(* PLC project marvel_vessel, Institute of Astronomy Onto 0.0.1 *)
(* stored: creationDateTime 2025-01-01T00:00:00.0, modificationDateTime 2025-01-01T00:00:00.0 *)

TYPE heaterControlProcesses : STRUCT
  {attribute 'TcHmiSymbol.Show'}
  start : Process;  (* Start warming up *)
  {attribute 'TcHmiSymbol.Show'}
  stop : Process;  (* Stop heating *)
  {attribute 'TcHmiSymbol.Show'}
  reset : Process;  (* Reset any errors *)
END_STRUCT;
END_TYPE

TYPE vesselProcesses : STRUCT
  {attribute 'TcHmiSymbol.Show'}
  initialize : Process;  (* Start initializing *)
  {attribute 'TcHmiSymbol.Show'}
  start : Process;  (* Start warming up *)
  {attribute 'TcHmiSymbol.Show'}
  stop : Process;  (* Stop all temperature control and heating *)
  {attribute 'TcHmiSymbol.Show'}
  reset : Process;  (* Reset any errors *)
END_STRUCT;
END_TYPE

TYPE temperatureMeasurementStatuses : STRUCT
  {attribute 'OPC.UA.DA' := '1'}
  {attribute 'OPC.UA.DA.Access' := '1'}
  {attribute 'TcHmiSymbol.Show'}
  enabled : EnabledStatus;  (* Is the temperature being measured? *)
  {attribute 'OPC.UA.DA' := '1'}
  {attribute 'OPC.UA.DA.Access' := '1'}
  {attribute 'TcHmiSymbol.Show'}
  health : HealthStatus;  (* Is the measurement OK? *)
  {attribute 'OPC.UA.DA' := '1'}
  {attribute 'OPC.UA.DA.Access' := '1'}
  {attribute 'TcHmiSymbol.Show'}
  alarm : HiHiLoLoAlarmStatus;  (* Alarm status *)
END_STRUCT;
END_TYPE

TYPE heaterControlStatuses : STRUCT
  {attribute 'OPC.UA.DA' := '1'}
  {attribute 'OPC.UA.DA.Access' := '1'}
  {attribute 'TcHmiSymbol.Show'}
  enabled : EnabledStatus;  (* Is the heater enabled? *)
  {attribute 'OPC.UA.DA' := '1'}
  {attribute 'OPC.UA.DA.Access' := '1'}
  {attribute 'TcHmiSymbol.Show'}
  health : HealthStatus;  (* Is the heater healthy? *)
  {attribute 'OPC.UA.DA' := '1'}
  {attribute 'OPC.UA.DA.Access' := '1'}
  {attribute 'TcHmiSymbol.Show'}
  busy : BusyStatus;  (* Is the heater busy (e.g. ramping)? *)
END_STRUCT;
END_TYPE

TYPE vesselStatuses : STRUCT
  {attribute 'OPC.UA.DA' := '1'}
  {attribute 'OPC.UA.DA.Access' := '1'}
  {attribute 'TcHmiSymbol.Show'}
  init : InitializationStatus;
  {attribute 'OPC.UA.DA' := '1'}
  {attribute 'OPC.UA.DA.Access' := '1'}
  {attribute 'TcHmiSymbol.Show'}
  health : HealthStatus;
  {attribute 'OPC.UA.DA' := '1'}
  {attribute 'OPC.UA.DA.Access' := '1'}
  {attribute 'TcHmiSymbol.Show'}
  busy : BusyStatus;
END_STRUCT;
END_TYPE

TYPE vesselHeaterConfig : STRUCT
  {attribute 'TcHmiSymbol.Show'}
  name : STRING;  (* Name of the heater *)
  {attribute 'TcHmiSymbol.Show'}
  enabled : BOOL;  (* True if the heater is enabled *)
  {attribute 'TcHmiSymbol.Show'}
  setPoint : REAL;  (* set point temperature in kelvin *)
  {attribute 'TcHmiSymbol.Show'}
  fastHeatingSetPoint : REAL;  (* set point temperature in kelvin used for fast heating (e.g. during ramping) *)
  {attribute 'TcHmiSymbol.Show'}
  maxPower : REAL;  (* Maximum power of the heater *)
  {attribute 'TcHmiSymbol.Show'}
  p : REAL;  (* proportional gain *)
  {attribute 'TcHmiSymbol.Show'}
  i : REAL;  (* integral gain *)
  {attribute 'TcHmiSymbol.Show'}
  d : REAL;  (* derivative gain *)
  {attribute 'TcHmiSymbol.Show'}
  weightTemperatureSensors : ARRAY[0..25] OF REAL;  (* value between 0-1 representing the weight of each temperature sensor (0 for sensors not effecting this heater) *)
END_STRUCT;
END_TYPE

TYPE vesselTemperatureSensorConfig : STRUCT
  {attribute 'TcHmiSymbol.Show'}
  name : STRING;  (* Name of the temperature sensor *)
  {attribute 'TcHmiSymbol.Show'}
  enabled : BOOL;  (* Is the quantity being measured? (Can be false e.g. if the sensor is deliberately not connected (yet).) *)
  {attribute 'TcHmiSymbol.Show'}
  gain : LREAL := 1.0;  (* Gain to be applied to the measured value (default: 1 = no gain) *)
  {attribute 'TcHmiSymbol.Show'}
  offset : LREAL;  (* Offset to be added to the measured value (default: 0 = no offset) *)
  {attribute 'TcHmiSymbol.Show'}
  alarms : HiHiLoLoAlarmConfig;  (* Config *)
END_STRUCT;
END_TYPE

TYPE vesselConfig : STRUCT
  {attribute 'TcHmiSymbol.Show'}
  setPointTarger : REAL;  (* set point temperature in kelvin *)
  {attribute 'TcHmiSymbol.Show'}
  rampVeloPos : REAL;  (* velocity of temperature change in K/s while ramping up *)
  {attribute 'TcHmiSymbol.Show'}
  rampVeloNeg : REAL;  (* velocity of temperature change in K/s while ramping down *)
END_STRUCT;
END_TYPE

TYPE M_SM_temperatureMeasurement : STRUCT
  {attribute 'OPC.UA.DA' := '1'}
  {attribute 'OPC.UA.DA.Access' := '1'}
  {attribute 'TcHmiSymbol.Show'}
  actualStatus : STRING;
  {attribute 'OPC.UA.DA' := '1'}
  {attribute 'OPC.UA.DA.Access' := '1'}
  {attribute 'TcHmiSymbol.Show'}
  actual : Temperature;
  {attribute 'OPC.UA.DA' := '1'}
  {attribute 'OPC.UA.DA.Access' := '1'}
  {attribute 'TcHmiSymbol.Show'}
  average : Temperature;
  {attribute 'OPC.UA.DA' := '1'}
  {attribute 'OPC.UA.DA.Access' := '1'}
  {attribute 'TcHmiSymbol.Show'}
  underrange : BOOL;
  {attribute 'OPC.UA.DA' := '1'}
  {attribute 'OPC.UA.DA.Access' := '1'}
  {attribute 'TcHmiSymbol.Show'}
  overrange : BOOL;
  {attribute 'OPC.UA.DA' := '1'}
  {attribute 'TcHmiSymbol.Show'}
  stat : temperatureMeasurementStatuses;
END_STRUCT;
END_TYPE

TYPE M_SM_heaterControl : STRUCT
  {attribute 'OPC.UA.DA' := '1'}
  {attribute 'OPC.UA.DA.Access' := '1'}
  {attribute 'TcHmiSymbol.Show'}
  actualStatus : STRING;
  {attribute 'OPC.UA.DA' := '1'}
  {attribute 'OPC.UA.DA.Access' := '1'}
  {attribute 'TcHmiSymbol.Show'}
  setPointRamped : REAL;
  {attribute 'OPC.UA.DA' := '1'}
  {attribute 'OPC.UA.DA.Access' := '1'}
  {attribute 'TcHmiSymbol.Show'}
  power : REAL;
  {attribute 'OPC.UA.DA' := '1'}
  {attribute 'OPC.UA.DA.Access' := '1'}
  {attribute 'TcHmiSymbol.Show'}
  associatedTemperature : REAL;
  {attribute 'OPC.UA.DA' := '1'}
  {attribute 'OPC.UA.DA.Access' := '1'}
  {attribute 'TcHmiSymbol.Show'}
  setPointDeviation : REAL;
  {attribute 'OPC.UA.DA' := '1'}
  {attribute 'OPC.UA.DA.Access' := '1'}
  {attribute 'TcHmiSymbol.Show'}
  isControlled : BOOL;
  {attribute 'OPC.UA.DA' := '1'}
  {attribute 'TcHmiSymbol.Show'}
  stat : heaterControlStatuses;
  {attribute 'OPC.UA.DA' := '1'}
  {attribute 'TcHmiSymbol.Show'}
  proc : M_SM_heaterControlProcesses;
END_STRUCT;
END_TYPE

TYPE M_SM_vessel : STRUCT
  {attribute 'OPC.UA.DA' := '1'}
  {attribute 'OPC.UA.DA.Access' := '1'}
  {attribute 'TcHmiSymbol.Show'}
  actualStatus : STRING;
  {attribute 'OPC.UA.DA' := '1'}
  {attribute 'OPC.UA.DA.Access' := '1'}
  {attribute 'TcHmiSymbol.Show'}
  config : vesselConfig;
  {attribute 'OPC.UA.DA' := '1'}
  {attribute 'OPC.UA.DA.Access' := '1'}
  {attribute 'TcHmiSymbol.Show'}
  isControlled : BOOL;
  {attribute 'OPC.UA.DA' := '1'}
  {attribute 'OPC.UA.DA.Access' := '1'}
  {attribute 'TcHmiSymbol.Show'}
  setPointRamped : REAL;
  {attribute 'OPC.UA.DA' := '1'}
  {attribute 'OPC.UA.DA.Access' := '1'}
  {attribute 'TcHmiSymbol.Show'}
  temperatureSensor : ARRAY[0..25] OF temperatureMeasurement;
  {attribute 'OPC.UA.DA' := '1'}
  {attribute 'OPC.UA.DA.Access' := '1'}
  {attribute 'TcHmiSymbol.Show'}
  vesselHeater : ARRAY[0..25] OF heaterControl;
  {attribute 'OPC.UA.DA' := '1'}
  {attribute 'TcHmiSymbol.Show'}
  stat : vesselStatuses;
  {attribute 'OPC.UA.DA' := '1'}
  {attribute 'TcHmiSymbol.Show'}
  proc : M_SM_vesselProcesses;
END_STRUCT;
END_TYPE

TYPE M_SM_heaterControlProcesses : STRUCT
  {attribute 'TcHmiSymbol.Show'}
  start : M_Process;
  {attribute 'TcHmiSymbol.Show'}
  stop : M_Process;
  {attribute 'TcHmiSymbol.Show'}
  reset : M_Process;
END_STRUCT;
END_TYPE

TYPE M_SM_vesselProcesses : STRUCT
  {attribute 'TcHmiSymbol.Show'}
  initialize : M_Process;
  {attribute 'TcHmiSymbol.Show'}
  start : M_Process;
  {attribute 'TcHmiSymbol.Show'}
  stop : M_Process;
  {attribute 'TcHmiSymbol.Show'}
  reset : M_Process;
END_STRUCT;
END_TYPE

FUNCTION_BLOCK SM_temperatureMeasurement
  VAR_INPUT
    {attribute 'OPC.UA.DA' := '0'}
    rawValue AT %I* : INT;  (* Measured raw value *)
    {attribute 'OPC.UA.DA' := '0'}
    error AT %I* : BOOL;  (* Error *)
    {attribute 'OPC.UA.DA' := '0'}
    conversionFactor : LREAL := 0.01;  (* rawValue * conversionFactor = temperature.degrees.value *)
  END_VAR
  VAR_OUTPUT
    {attribute 'OPC.UA.DA' := '1'}
    {attribute 'OPC.UA.DA.Access' := '1'}
    actualStatus : STRING(50);  (* Current status description *)
    {attribute 'OPC.UA.DA' := '1'}
    {attribute 'OPC.UA.DA.Access' := '1'}
    actual : Temperature;  (* Actual value *)
    {attribute 'OPC.UA.DA' := '1'}
    {attribute 'OPC.UA.DA.Access' := '1'}
    average : Temperature;  (* Moving average value *)
    {attribute 'OPC.UA.DA' := '1'}
    {attribute 'OPC.UA.DA.Access' := '1'}
    underrange AT %I* : BOOL;  (* Underrange *)
    {attribute 'OPC.UA.DA' := '1'}
    {attribute 'OPC.UA.DA.Access' := '1'}
    overrange AT %I* : BOOL;  (* Overrange *)
    {attribute 'OPC.UA.DA' := '1'}
    stat : temperatureMeasurementStatuses;  (* Statuses of the state machine *)
  END_VAR
  VAR_IN_OUT
    {attribute 'OPC.UA.DA' := '0'}
    config : vesselTemperatureSensorConfig;  (* Reference to the config (alarms in degrees celsius) *)
    {attribute 'OPC.UA.DA' := '0'}
    activity_ref : ActivityStatus;  (* Shared activity status *)
    {attribute 'OPC.UA.DA' := '0'}
    services_ref : Services;  (* Shared services *)
  END_VAR

            stat.enabled := F_EnabledStatus(
    superState := TRUE,
    isEnabled := config.enabled);
stat.health := F_HealthStatus(
    superState := stat.enabled = EnabledStatus.enabled,
    isGood := NOT(error OR (underrange OR (overrange OR ((stat.alarm = HiHiLoLoAlarmStatus.hiHi) OR (stat.alarm = HiHiLoLoAlarmStatus.loLo))))),
    hasWarning := (stat.alarm = HiHiLoLoAlarmStatus.hi) OR (stat.alarm = HiHiLoLoAlarmStatus.lo));
stat.alarm := F_HiHiLoLoAlarmStatus(
    superState := stat.enabled = EnabledStatus.enabled,
    config := config.alarms,
    value := average.celsius.value);

          

METHOD _copyFromModel_SM_temperatureMeasurement
  VAR_IN_OUT
    {attribute 'OPC.UA.DA' := '0'}
    model : M_SM_temperatureMeasurement;
  END_VAR
                  
                
END_METHOD

METHOD _copyToModel_SM_temperatureMeasurement
  VAR_IN_OUT
    {attribute 'OPC.UA.DA' := '0'}
    model : M_SM_temperatureMeasurement;
  END_VAR
                  model.actualStatus := THIS^.actualStatus;
model.actual := THIS^.actual;
model.average := THIS^.average;
model.underrange := THIS^.underrange;
model.overrange := THIS^.overrange;
model.stat := THIS^.stat;

                
END_METHOD
END_FUNCTION_BLOCK

FUNCTION_BLOCK SM_heaterControl
  VAR_OUTPUT
    {attribute 'OPC.UA.DA' := '1'}
    {attribute 'OPC.UA.DA.Access' := '1'}
    actualStatus : STRING(50);  (* Current status description *)
    {attribute 'OPC.UA.DA' := '1'}
    {attribute 'OPC.UA.DA.Access' := '1'}
    setPointRamped : REAL;  (* Set point temperature in kelvin *)
    {attribute 'OPC.UA.DA' := '1'}
    {attribute 'OPC.UA.DA.Access' := '1'}
    power : REAL;  (* Current power of the heater in percentage *)
    {attribute 'OPC.UA.DA' := '1'}
    {attribute 'OPC.UA.DA.Access' := '1'}
    associatedTemperature : REAL;  (* Temperature associated with the heater *)
    {attribute 'OPC.UA.DA' := '1'}
    {attribute 'OPC.UA.DA.Access' := '1'}
    setPointDeviation : REAL;  (* Current error between set point and associated temperature *)
    {attribute 'OPC.UA.DA' := '1'}
    {attribute 'OPC.UA.DA.Access' := '1'}
    isControlled : BOOL;  (* True if the heater is in controlled state *)
    {attribute 'OPC.UA.DA' := '1'}
    stat : heaterControlStatuses;  (* Statuses of the state machine *)
    {attribute 'OPC.UA.DA' := '1'}
    proc : heaterControlProcesses;  (* Processes of the state machine *)
  END_VAR
  VAR_IN_OUT
    {attribute 'OPC.UA.DA' := '0'}
    config : vesselHeaterConfig;  (* Reference to the heater config *)
    {attribute 'OPC.UA.DA' := '0'}
    activity_ref : ActivityStatus;  (* Shared activity status *)
    {attribute 'OPC.UA.DA' := '0'}
    services_ref : Services;  (* Shared services *)
  END_VAR

            stat.enabled := F_EnabledStatus(
    superState := TRUE,
    isEnabled := config.enabled);
stat.health := F_HealthStatus( superState := TRUE );
stat.busy := F_BusyStatus(
    superState := TRUE,
    isBusy := proc.start.stat.busy);
proc.start( isEnabled := config.enabled );
proc.stop();
proc.reset();

          

METHOD _copyFromModel_SM_heaterControl
  VAR_IN_OUT
    {attribute 'OPC.UA.DA' := '0'}
    model : M_SM_heaterControl;
  END_VAR
                  THIS^.proc.start._copyFromModel_Process( model := model.proc.start );
THIS^.proc.stop._copyFromModel_Process( model := model.proc.stop );
THIS^.proc.reset._copyFromModel_Process( model := model.proc.reset );

                
END_METHOD

METHOD _copyToModel_SM_heaterControl
  VAR_IN_OUT
    {attribute 'OPC.UA.DA' := '0'}
    model : M_SM_heaterControl;
  END_VAR
                  model.actualStatus := THIS^.actualStatus;
model.setPointRamped := THIS^.setPointRamped;
model.power := THIS^.power;
model.associatedTemperature := THIS^.associatedTemperature;
model.setPointDeviation := THIS^.setPointDeviation;
model.isControlled := THIS^.isControlled;
model.stat := THIS^.stat;
THIS^.proc.start._copyToModel_Process( model := model.proc.start );
THIS^.proc.stop._copyToModel_Process( model := model.proc.stop );
THIS^.proc.reset._copyToModel_Process( model := model.proc.reset );

                
END_METHOD
END_FUNCTION_BLOCK

FUNCTION_BLOCK SM_vessel
  VAR_OUTPUT
    {attribute 'OPC.UA.DA' := '1'}
    {attribute 'OPC.UA.DA.Access' := '1'}
    actualStatus : STRING(50);  (* Current status description *)
    {attribute 'OPC.UA.DA' := '1'}
    {attribute 'OPC.UA.DA.Access' := '1'}
    config : vesselConfig;  (* Active configuration of the vessel *)
    {attribute 'OPC.UA.DA' := '1'}
    {attribute 'OPC.UA.DA.Access' := '1'}
    isControlled : BOOL;  (* True if the vessel is in controlled state *)
    {attribute 'OPC.UA.DA' := '1'}
    {attribute 'OPC.UA.DA.Access' := '1'}
    setPointRamped : REAL;  (* Set point temperature in kelvin after ramping *)
    {attribute 'OPC.UA.DA' := '1'}
    {attribute 'OPC.UA.DA.Access' := '1'}
    temperatureSensor : ARRAY[0..25] OF temperatureMeasurement;  (* All vessel temperature sensors *)
    {attribute 'OPC.UA.DA' := '1'}
    {attribute 'OPC.UA.DA.Access' := '1'}
    vesselHeater : ARRAY[0..25] OF heaterControl;  (* All vessel heaters *)
    {attribute 'OPC.UA.DA' := '1'}
    stat : vesselStatuses;  (* Statuses of the state machine *)
    {attribute 'OPC.UA.DA' := '1'}
    proc : vesselProcesses;  (* Processes of the state machine *)
  END_VAR
  VAR_IN_OUT
    {attribute 'OPC.UA.DA' := '0'}
    activity_ref : ActivityStatus;  (* Shared activity status *)
    {attribute 'OPC.UA.DA' := '0'}
    services_ref : Services;  (* Shared services *)
    {attribute 'OPC.UA.DA' := '0'}
    config_ref : vesselConfig;  (* Active configuration of the vessel *)
  END_VAR

            stat.health := F_HealthStatus(
    superState := TRUE,
    isGood := ((stat.health = HealthStatus.good) OR (stat.health = HealthStatus.warning)) AND ((stat.health = HealthStatus.good) OR (stat.health = HealthStatus.warning)));
proc.initialize( isEnabled := (NOT(stat.init = InitializationStatus.locked)) AND ((stat.init = InitializationStatus.shutdown) OR ((stat.init = InitializationStatus.initializingFailed) OR (stat.init = InitializationStatus.initialized))) );
proc.start( isEnabled := (stat.init = InitializationStatus.initializingFailed) AND (stat.init = InitializationStatus.initialized) );
proc.stop( isEnabled := (stat.busy = BusyStatus.busy) OR isControlled );
proc.reset( isEnabled := (stat.busy = BusyStatus.idle) AND (stat.init = InitializationStatus.initialized) );

          

METHOD _copyFromModel_SM_vessel
  VAR_IN_OUT
    {attribute 'OPC.UA.DA' := '0'}
    model : M_SM_vessel;
  END_VAR
                  THIS^.proc.initialize._copyFromModel_Process( model := model.proc.initialize );
THIS^.proc.start._copyFromModel_Process( model := model.proc.start );
THIS^.proc.stop._copyFromModel_Process( model := model.proc.stop );
THIS^.proc.reset._copyFromModel_Process( model := model.proc.reset );

                
END_METHOD

METHOD _copyToModel_SM_vessel
  VAR_IN_OUT
    {attribute 'OPC.UA.DA' := '0'}
    model : M_SM_vessel;
  END_VAR
                  model.actualStatus := THIS^.actualStatus;
model.config := THIS^.config;
model.isControlled := THIS^.isControlled;
model.setPointRamped := THIS^.setPointRamped;
model.temperatureSensor := THIS^.temperatureSensor;
model.vesselHeater := THIS^.vesselHeater;
model.stat := THIS^.stat;
THIS^.proc.initialize._copyToModel_Process( model := model.proc.initialize );
THIS^.proc.start._copyToModel_Process( model := model.proc.start );
THIS^.proc.stop._copyToModel_Process( model := model.proc.stop );
THIS^.proc.reset._copyToModel_Process( model := model.proc.reset );

                
END_METHOD
END_FUNCTION_BLOCK
